(* IEC 61131-3 sources: plc_generation_empirical_study/datasets/task_bank_c06_bounded_runtime_v0_3/tasks/C06_U19_lean_composite, 2 files *)

(* ---- interface.st ---- *)
FUNCTION_BLOCK C06_U19_lean_composite
VAR_INPUT
    A_AddItem : BOOL;
    A_RemoveItem : BOOL;
    A_Reset : BOOL;
    A_Capacity : INT;
    B_AutoMode : BOOL;
    B_AutoDemand : BOOL;
    B_ManualDemand : BOOL;
    B_SafetyOK : BOOL;
    B_Inhibit : BOOL;
    SubsystemBEnable : BOOL;
    CrossReset : BOOL;
END_VAR
VAR_OUTPUT
    A_Count : INT;
    A_Empty : BOOL;
    A_Full : BOOL;
    A_Conflict : BOOL;
    B_Command : BOOL;
    B_Blocked : BOOL;
    CrossReady : BOOL;
    CrossBlocked : BOOL;
END_VAR
END_FUNCTION_BLOCK

(* ---- reference.st ---- *)
FUNCTION_BLOCK C06_U19_lean_composite
VAR_INPUT
    A_AddItem : BOOL;
    A_RemoveItem : BOOL;
    A_Reset : BOOL;
    A_Capacity : INT;
    B_AutoMode : BOOL;
    B_AutoDemand : BOOL;
    B_ManualDemand : BOOL;
    B_SafetyOK : BOOL;
    B_Inhibit : BOOL;
    SubsystemBEnable : BOOL;
    CrossReset : BOOL;
END_VAR
VAR_OUTPUT
    A_Count : INT;
    A_Empty : BOOL;
    A_Full : BOOL;
    A_Conflict : BOOL;
    B_Command : BOOL;
    B_Blocked : BOOL;
    CrossReady : BOOL;
    CrossBlocked : BOOL;
END_VAR
VAR
    A_PrevAdd : BOOL := FALSE;
    A_PrevRemove : BOOL := FALSE;
END_VAR

A_Conflict := FALSE;
IF A_Reset THEN
    A_Count := 0;
ELSIF A_AddItem AND (NOT A_PrevAdd) AND A_RemoveItem AND (NOT A_PrevRemove) THEN
    A_Conflict := TRUE;
ELSIF A_AddItem AND (NOT A_PrevAdd) AND (A_Count < A_Capacity) THEN
    A_Count := A_Count + 1;
ELSIF A_RemoveItem AND (NOT A_PrevRemove) AND (A_Count > 0) THEN
    A_Count := A_Count - 1;
END_IF;
A_Empty := A_Count = 0;
A_Full := A_Count >= A_Capacity;
A_PrevAdd := A_AddItem;
A_PrevRemove := A_RemoveItem;

IF CrossReset THEN
    CrossReady := FALSE;
ELSIF A_Empty THEN
    CrossReady := TRUE;
END_IF;
CrossBlocked := SubsystemBEnable AND (NOT CrossReady);

IF SubsystemBEnable AND CrossReady THEN
    B_Command := ((B_AutoMode AND B_AutoDemand) OR ((NOT B_AutoMode) AND B_ManualDemand))
               AND B_SafetyOK AND (NOT B_Inhibit);
    B_Blocked := ((B_AutoMode AND B_AutoDemand) OR ((NOT B_AutoMode) AND B_ManualDemand))
               AND ((NOT B_SafetyOK) OR B_Inhibit);
ELSE
    B_Command := FALSE;
    B_Blocked := FALSE;
END_IF;

END_FUNCTION_BLOCK
